# EPICS substitutions: iocs/mcf01/ppmacApp/Db/pmacStatus.substitutions
file "db/ppmacStatus.db"
{
pattern
{SYS,               PMAC,    VERSION  PLC  PORT,  NAXES }
{"XF:27IDF-CT",     "MC:01", "1"      5    "P0",  8     }
}
